PROGRAM LogicalCircuits_Ex07
VAR
	S1					: DigitalInput_NO;
	S2					: DigitalInput_NC;
	P1 					: DigitalOutput;
END_VAR

IF S1.isOn OR S2.broken THEN
	P1.On();
END_IF

END_PROGRAM

(* stored: Version 1.1.0.1
   POU LogicalCircuits_Ex07: Id {b368deaa-c957-47b2-aaf7-460a78b7acef}, SpecialFunc None *)
